// Implicitly generated code : DO NOT EDIT
FUNCTION CheckLRangeUnsigned : ULINT
VAR_INPUT
	value, lower, upper: ULINT;
END_VAR

// Implicitly generated code : Only an Implementation suggestion
{noflow}
IF (value < lower) THEN
	CheckLRangeUnsigned := lower;
ELSIF(value > upper) THEN
	CheckLRangeUnsigned := upper;
ELSE
	CheckLRangeUnsigned := value;
END_IF
{flow}

END_FUNCTION

(* stored: Version 1.1.0.1, ProductVersion 3.1.4024.4
   POU CheckLRangeUnsigned: Id {aa02d5f5-a960-4cf4-86a0-c35ae72406d2}, SpecialFunc CheckLRangeUnsigned *)
